(* IEC 61131-3 sources: ae-motion-tiax/src, 2 files *)

(* ---- library.st ---- *)
NAMESPACE SimaticAx.Lib

    CLASS PUBLIC ControlAxis
        VAR PRIVATE
            _started : BOOL;
        END_VAR

        VAR PRIVATE

        END_VAR

        METHOD PUBLIC Enable : BOOL
            // TODO implement
            Enable := TRUE;
        END_METHOD

        METHOD PUBLIC Move : BOOL
            VAR_INPUT
                speed : LREAL;
            END_VAR
            // TODO implement
            Move := TRUE;
        END_METHOD

        METHOD PUBLIC Stop : BOOL
            // TODO implement
            Stop := TRUE;
        END_METHOD

    END_CLASS

END_NAMESPACE

(* ---- wrapper.st ---- *)
NAMESPACE SimaticAx.Lib

    FUNCTION_BLOCK MotorWrapper
        VAR_INPUT
            start : BOOL;
        END_VAR
        VAR
            m : ControlAxis;
        END_VAR

        IF start THEN
            m.Enable();
        END_IF;
    END_FUNCTION_BLOCK

END_NAMESPACE
